{attribute 'hide_all_locals'}
FUNCTION_BLOCK TemperatureArgument IMPLEMENTS I_SimpleLogArgument
VAR
	_SetPoint : LREAL;
	_Actual	  : LREAL;
END_VAR

{attribute 'monitoring':='call'}
PROPERTY ActualTemperature : LREAL
GET
ActualTemperature := _Actual;
END_GET
SET
_Actual := ActualTemperature;
END_SET
END_PROPERTY

{attribute 'monitoring':='call'}
PROPERTY SetPoint : LREAL
GET
SetPoint := _SetPoint;
END_GET
SET
_SetPoint := SetPoint;
END_SET
END_PROPERTY

METHOD ToString : T_MaxString
ToString := Concat('Set Temperature: ', CONCAT(TO_STRING(_SetPoint), CONCAT(' , Actual Temp: ', TO_STRING(_Actual))));
END_METHOD

END_FUNCTION_BLOCK

(* stored: Version 1.1.0.1
   POU TemperatureArgument: Id {b3a135e7-6ead-4b8c-99f7-8a4ced55e20a}, SpecialFunc None
   Property ActualTemperature: Id {559f96be-b291-4b99-9c53-b1e995b43457}
   Get Get: Id {939a2349-97de-4f35-a2f2-e341a10edbf3}
   Set Set: Id {ff7da045-ab2a-4144-96ac-6882f872fb27}
   Property SetPoint: Id {5fbd6915-084d-402c-893c-77076ef0a69c}
   Get Get: Id {38d870af-c045-4f70-b98d-43f9efed54b0}
   Set Set: Id {ec1d1361-9581-4566-a382-a56aeaffbaa1}
   Method ToString: Id {a6d0c48e-0953-4c20-af52-a513215bcbc1} *)
